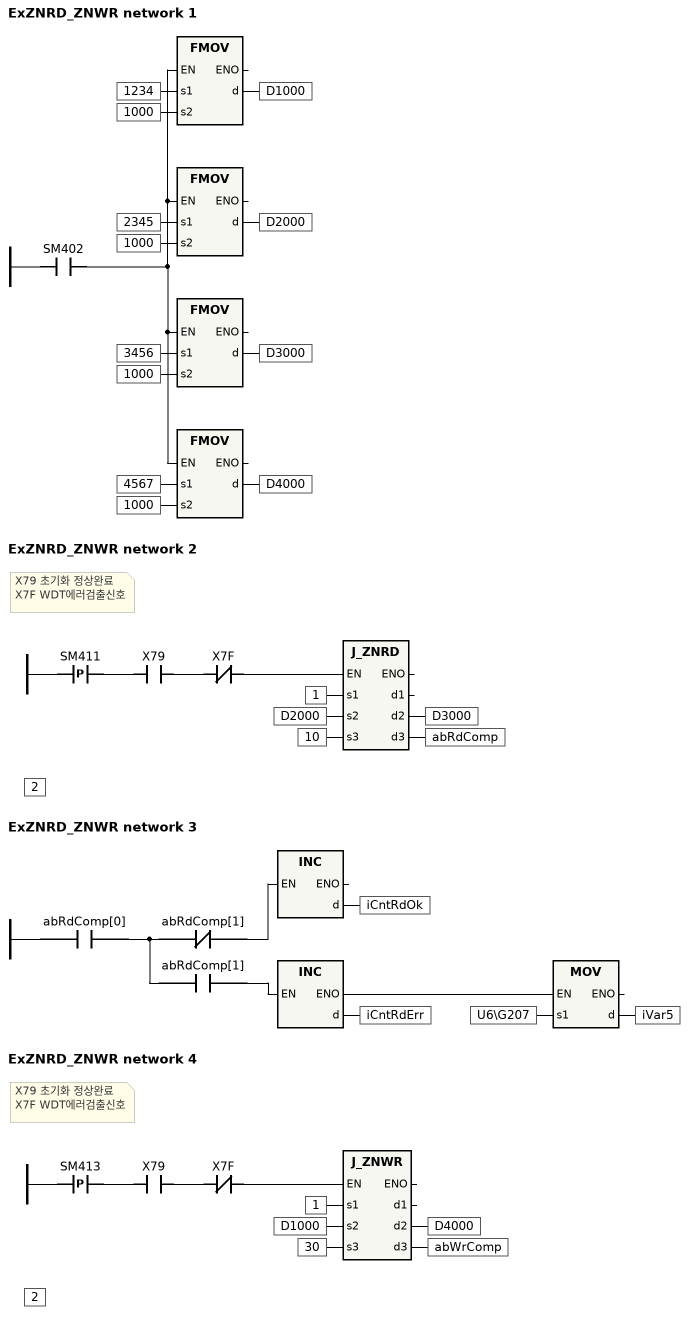
(* [picture p24: structured ladder/FBD of ExZNRD_ZNWR, networks 1 to 4] *)
(* network 1 *)
FMOV(SM402, 1234, 1000, D1000);
FMOV(SM402, 2345, 1000, D2000);
FMOV(SM402, 3456, 1000, D3000);
FMOV(SM402, 4567, 1000, D4000);
(* network 2 *)
(* X79 초기화 정상완료 / X7F WDT에러검출신호 *)
J_ZNRD(LDP(TRUE, SM411) AND X79 AND NOT X7F, 1, D2000, 10, _open, D3000, abRdComp);
(* not connected to any output: 2 *)
(* network 3 *)
INC(abRdComp[0] AND NOT abRdComp[1], iCntRdOk);
_e1 := INC(abRdComp[0] AND abRdComp[1], iCntRdErr);
MOV(_e1, U6\G207, iVar5);
(* network 4 *)
(* X79 초기화 정상완료 / X7F WDT에러검출신호 *)
J_ZNWR(LDP(TRUE, SM413) AND X79 AND NOT X7F, 1, D1000, 30, _open, D4000, abWrComp);
(* not connected to any output: 2 *)
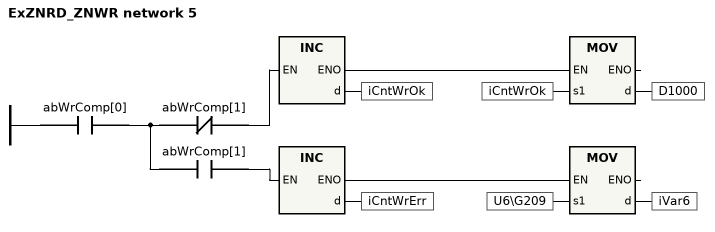
(* network 5 *)
_e1 := INC(abWrComp[0] AND NOT abWrComp[1], iCntWrOk);
MOV(_e1, iCntWrOk, D1000);
_e2 := INC(abWrComp[0] AND abWrComp[1], iCntWrErr);
MOV(_e2, U6\G209, iVar6);
END_PROGRAM
